// TIA Portal V18 export
TYPE "LGasp_typeArticolo"
// stored: IsFailsafeCompliant false
   STRUCT
      general : "LGasp_typeArticoloGenerale";   // generale
      prepunchingquota : Array[1.."NumPunzonateArticolo"] of "LGasp_typeQuota";   // quote prepunzonatura
   END_STRUCT;
END_TYPE
